// TIA Portal V20 export
// export: Created 2025-12-01T14:57:20.1582824Z, ExportSetting None, DisplayName Totally Integrated Automation Portal, DisplayVersion V20 Update 3, DisplayName TIA Portal Openness, DisplayVersion V20 Update 3, DisplayName TIA Portal Version Control Interface, DisplayVersion V20 Update 3, DisplayName STEP 7 Professional, DisplayVersion V20 Update 3, DisplayName STEP 7 Safety, DisplayVersion V20 Update 2, DisplayName WinCC Basic/Comfort/Advanced, DisplayVersion V20 Update 3, DisplayName WinCC Professional, DisplayVersion V20 Update 3, DisplayName WinCC Unified, DisplayVersion V20 Update 3
DATA_BLOCK "DB860_Bits_ErroresArmarios"   // DB860
{ S7_Optimized_Access := 'FALSE' }
AUTHOR : ERRORES
NAME : 20131009
VERSION : 3.1
// stored: AutoNumber false
   VAR RETAIN
      Armarios : Array[0.."CTE_MaxDispositivos"] of Struct   // Variable provisional
         Emergencias : Array[0..15] of Bool;
         ErroresGraves : Array[0..15] of Bool;
         ErroresLeves : Array[0..95] of Bool;
      END_STRUCT;
   END_VAR
BEGIN
END_DATA_BLOCK
